{attribute addProperty BoxType "EL9540-0010-0016"}
{attribute addProperty Id "Status_UpAT %I*Status_Up_B12359DC1620WcStateAT %I*WcState_98A4DF7520.250InfoDataAT %I*InfoData_192954DE1620"}
{attribute addProperty CRC "2220945836"}
{attribute addProperty SizeInBites "34"}
{attribute addProperty SizeInBytes "4.25"}
TYPE EL9540_081B367B :
STRUCT
	{attribute addProperty Name "Status_Up"}
	Status_Up : Status_Up_B12359DC;
	{attribute addProperty Name "WcState"}
	WcState : WcState_98A4DF75;
	{attribute addProperty Name "InfoData"}
	InfoData : InfoData_192954DE;
END_STRUCT
END_TYPE

(* stored: Version 1.2.0.0, ProductVersion 3.1.4024.9
   DUT EL9540_081B367B: Id {82150e83-29d0-4c74-aedc-7885ff991546} *)
